(* Logix 5000 project; controller cal1615 1756-L62 rev 20.19; software revision 20.05; part 81 of 81 *)
(* tags used below, declared in another part *)
   A00 : ALIAS FOR hmi_dint[0].0;
   A01 : ALIAS FOR hmi_dint[0].1;
   A08 : ALIAS FOR hmi_dint[0].8;
   A12 : ALIAS FOR hmi_dint[0].12;
   A30 : ALIAS FOR hmi_dint[0].30;
   ai_lpt01_pct : REAL;   // AI: Linear Position Transducer [%]
   ao_prs02 : REAL;   // AO: Pressure 2
   do_close_nip_sol : ALIAS FOR p00_io_winder:4:O.8;
   do_nip_illuminated_ss : ALIAS FOR p00_io_winder:4:O.6;
   man_pos_active : ALIAS FOR hmi_dint[9].11;
   man_pos_at_position : ALIAS FOR hmi_dint[9].14;
   man_pos_err : REAL;   // Accumulator Manual Position Mode Absolute Position Error [% of Stroke]
   man_pos_pid : PID;   // Accumulator Manual Position Mode Position to Pressure PID
   man_pos_pid_cv : REAL;   // Accumulator Manual Position Mode PID Control Variable [psi]
   man_pos_pid_pv : REAL;   // Accumulator Manual Position Mode PID Process Variable [% of Stroke]
   man_pos_pressure : REAL;   // Accumulator Manual Position Mode Pressure Command [psi]
   man_pos_request : ALIAS FOR hmi_dint[9].9;
   man_pos_sp : REAL;   // Accumulator Manual Position Mode Setpoint in Use Operator Entry After Clamp [% of Stroke]
   man_pos_timer : TIMER;   // Accumulator Manual Position Mode PID Update Timer
   Me : ALIAS FOR p00_wac;
   nip_auto_open_request : BOOL;   // Nip Auto Open Request
   nip_close_request : ALIAS FOR hmi_dint[9].7;
   nip_mode_auto : BOOL;   // Nip Mode Auto
   nip_open_dwell : TIMER;   // Nip Roll Open Dwell Payout must be established before the nip lets go
   nip_open_request : BOOL;   // Nip Open Request
   oneshot : DINT;
   param_acc_min_limit : REAL;   // Parameter Accumulator Low Min Limimt
   param_man_pos_db : REAL;   // Parameter Manual Position Mode Hold Deadband At position and output frozen inside this band [% of Stroke]
   param_man_pos_kd : REAL;   // Parameter Manual Position Mode PID Rate Time Dependent gains form [min]
   param_man_pos_ki : REAL;   // Parameter Manual Position Mode PID Reset Time Dependent gains form, 0 = no integral [min per repeat]
   param_man_pos_kp : REAL;   // Parameter Manual Position Mode PID Controller Gain Dependent gains form [psi per % of Stroke]
   param_man_pos_prs_max : REAL;   // Parameter Manual Position Mode Pressure Command Upper Limit [psi]
   param_man_pos_prs_min : REAL;   // Parameter Manual Position Mode Pressure Command Lower Limit [psi]
   param_man_pos_sp : REAL;   // Parameter Manual Position Mode Target Carriage Position Operator Entry [% of Stroke]
   param_man_pos_sp_max : REAL;   // Parameter Manual Position Mode Highest Target Allowed Keeps the carriage off the full limit [% of Stroke]
   param_man_pos_sp_min : REAL;   // Parameter Manual Position Mode Lowest Target Allowed Keeps the carriage off the empty limit [% of Stroke]
   param_man_pos_upd_ms : DINT;   // Parameter Manual Position Mode PID Update Interval [ms]
   param_tare_pressure : REAL;   // Parameter Friction Trim Pressure Carriage Balanced - No Drift Up or Down Set at Installation
   pb_acc_on : ALIAS FOR hmi_dint[9].2;
   request_fill : ALIAS FOR hmi_dint[9].1;
   timer_nip_open_delay : TIMER;   // Nip Open Dwell Timer
   W00 : ALIAS FOR hmi_dint[2].0;
   winder_running : BOOL;   // Winder Running
   FAULT : BOOL;   // Fault AFI
   HMI : BOOL;   // AFI HMI
   nip_mode_close : BOOL;   // Nip Mode Close
   p00_FlashBit_1Sec : BOOL;   // System Flash Bit 1 Second
   p00_pb_lamp_test : BOOL;
   p01r09 : routine;   // System Modes
(* P31_WAC, continued *)

ROUTINE R23_Position_Control   (* ladder *)
// Windup Accumulator
// Manual Position Control
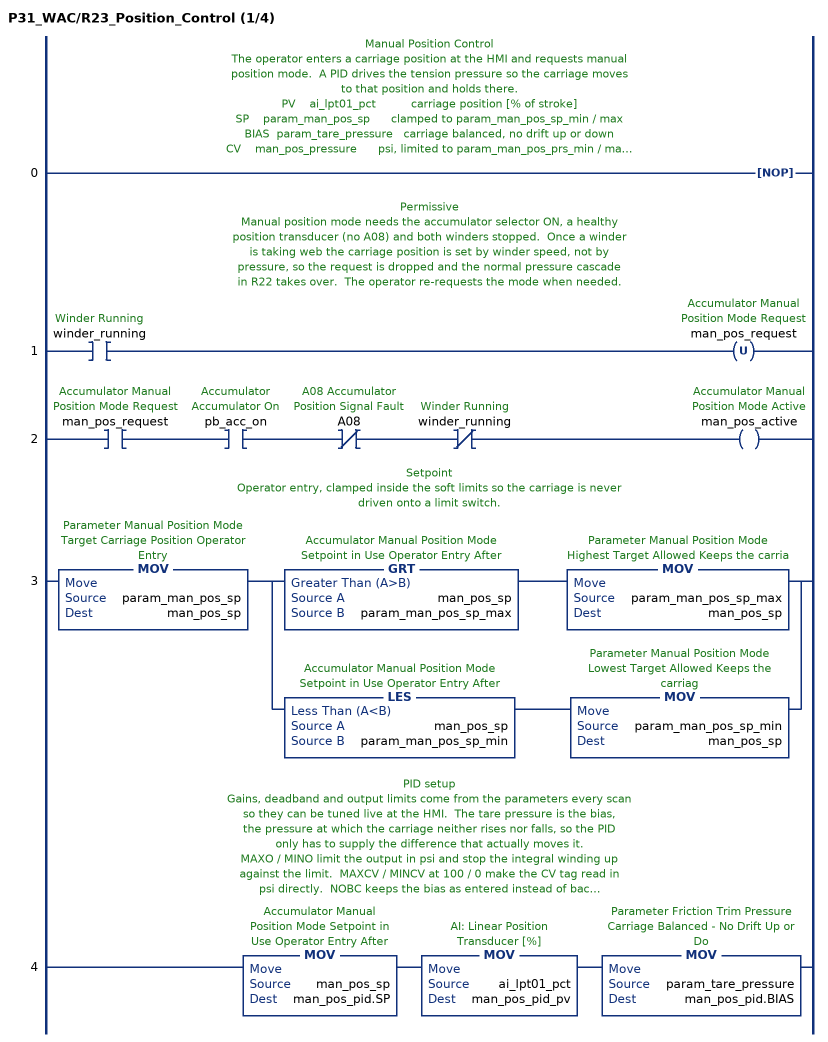
   // Manual Position Control
   // The operator enters a carriage position at the HMI and requests manual
   // position mode.  A PID drives the tension pressure so the carriage moves
   // to that position and holds there.
   //   PV    ai_lpt01_pct          carriage position [% of stroke]
   //   SP    param_man_pos_sp      clamped to param_man_pos_sp_min / max
   //   BIAS  param_tare_pressure   carriage balanced, no drift up or down
   //   CV    man_pos_pressure      psi, limited to param_man_pos_prs_min / max
   // Error = SP - PV.  Carriage below target -> more pressure -> carriage
   // rises.  Dependent gains form, the same as the P20 and P29 loops:
   // Kp in psi per % of stroke, Ki as reset time in minutes per repeat.
   // man_pos_pressure is picked up in R22 ahead of sys_Ramp, so the existing
   // accel/decel ramp still smooths the output.
   // Rev 20260923 a01
   0: NOP();
   // Permissive
   // Manual position mode needs the accumulator selector ON, a healthy
   // position transducer (no A08) and both winders stopped.  Once a winder
   // is taking web the carriage position is set by winder speed, not by
   // pressure, so the request is dropped and the normal pressure cascade
   // in R22 takes over.  The operator re-requests the mode when needed.
   1: XIC(winder_running)OTU(man_pos_request);
   2: XIC(man_pos_request)XIC(pb_acc_on)XIO(A08)XIO(winder_running)OTE(man_pos_active);
   // Setpoint
   // Operator entry, clamped inside the soft limits so the carriage is never
   // driven onto a limit switch.
   3: MOV(param_man_pos_sp,man_pos_sp)[GRT(man_pos_sp,param_man_pos_sp_max) MOV(param_man_pos_sp_max,man_pos_sp) ,LES(man_pos_sp,param_man_pos_sp_min) MOV(param_man_pos_sp_min,man_pos_sp) ];
   // PID setup
   // Gains, deadband and output limits come from the parameters every scan
   // so they can be tuned live at the HMI.  The tare pressure is the bias,
   // the pressure at which the carriage neither rises nor falls, so the PID
   // only has to supply the difference that actually moves it.
   // MAXO / MINO limit the output in psi and stop the integral winding up
   // against the limit.  MAXCV / MINCV at 100 / 0 make the CV tag read in
   // psi directly.  NOBC keeps the bias as entered instead of back
   // calculating it.  NOZC makes the deadband take effect as soon as the
   // error is inside it, so the carriage holds where it stops instead of
   // hunting for an exact zero crossing.
   4: MOV(man_pos_sp,man_pos_pid.SP)MOV(ai_lpt01_pct,man_pos_pid_pv)MOV(param_tare_pressure,man_pos_pid.BIAS);
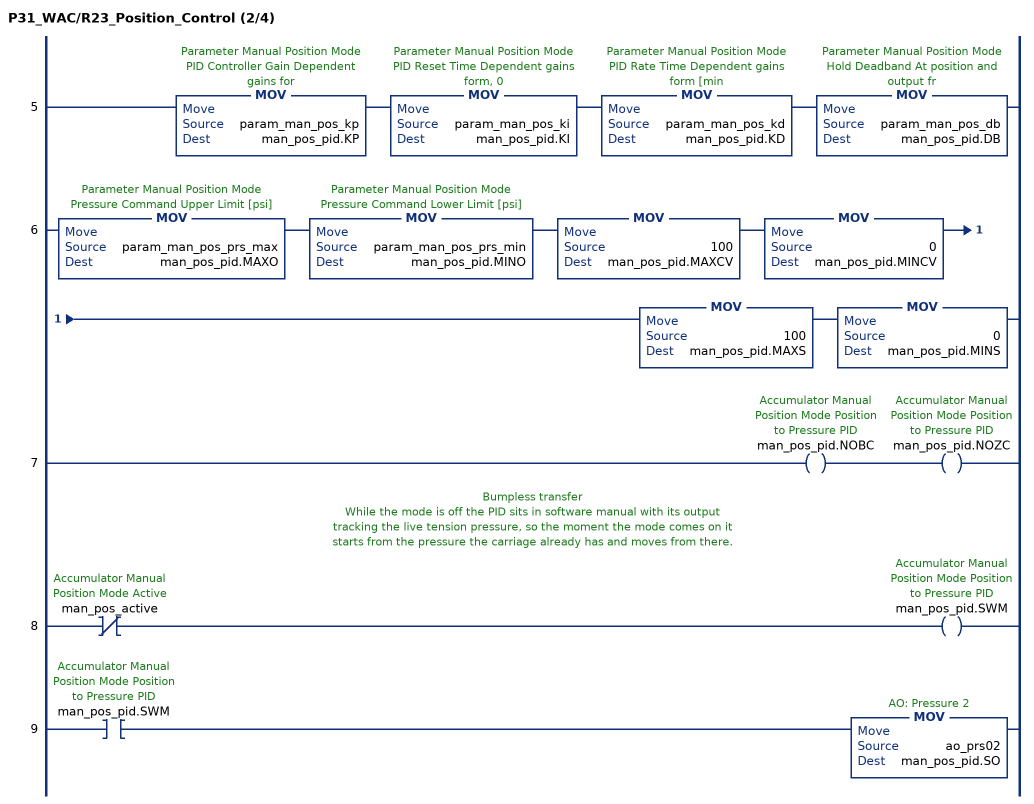
   5: MOV(param_man_pos_kp,man_pos_pid.KP)MOV(param_man_pos_ki,man_pos_pid.KI)MOV(param_man_pos_kd,man_pos_pid.KD)MOV(param_man_pos_db,man_pos_pid.DB);
   6: MOV(param_man_pos_prs_max,man_pos_pid.MAXO)MOV(param_man_pos_prs_min,man_pos_pid.MINO)MOV(100,man_pos_pid.MAXCV)MOV(0,man_pos_pid.MINCV)MOV(100,man_pos_pid.MAXS)MOV(0,man_pos_pid.MINS);
   7: OTE(man_pos_pid.NOBC)OTE(man_pos_pid.NOZC);
   // Bumpless transfer
   // While the mode is off the PID sits in software manual with its output
   // tracking the live tension pressure, so the moment the mode comes on it
   // starts from the pressure the carriage already has and moves from there.
   8: XIO(man_pos_active)OTE(man_pos_pid.SWM);
   9: XIC(man_pos_pid.SWM)MOV(ao_prs02,man_pos_pid.SO);
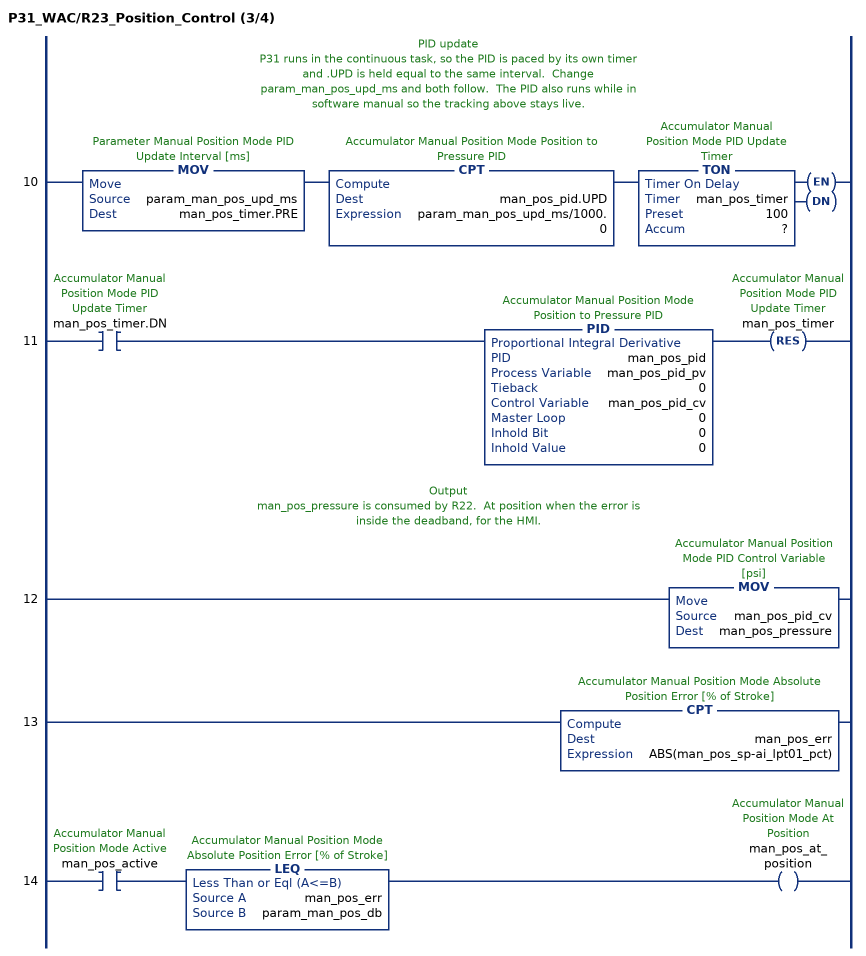
   // PID update
   // P31 runs in the continuous task, so the PID is paced by its own timer
   // and .UPD is held equal to the same interval.  Change
   // param_man_pos_upd_ms and both follow.  The PID also runs while in
   // software manual so the tracking above stays live.
   10: MOV(param_man_pos_upd_ms,man_pos_timer.PRE)CPT(man_pos_pid.UPD,param_man_pos_upd_ms/1000.0)TON(man_pos_timer,?,?);
   11: XIC(man_pos_timer.DN)PID(man_pos_pid,man_pos_pid_pv,0,man_pos_pid_cv,0,0,0)RES(man_pos_timer);
   // Output
   // man_pos_pressure is consumed by R22.  At position when the error is
   // inside the deadband, for the HMI.
   12: MOV(man_pos_pid_cv,man_pos_pressure);
   13: CPT(man_pos_err,ABS(man_pos_sp-ai_lpt01_pct));
   14: XIC(man_pos_active)LEQ(man_pos_err,param_man_pos_db)OTE(man_pos_at_position);
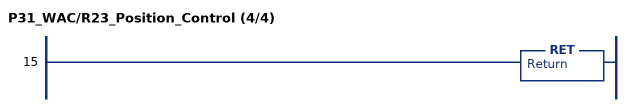
   15: RET();
END_ROUTINE

ROUTINE R31_Nip_Roll   (* ladder *)
// WAC
// Nip Roll
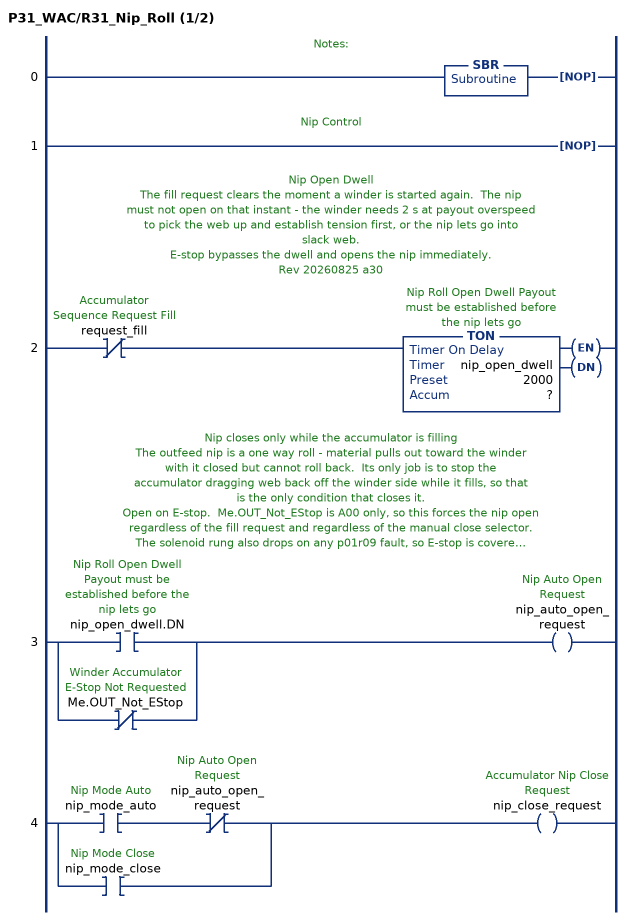
   // Notes:
   0: SBR()NOP();
   // Nip Control
   1: NOP();
   // Nip Open Dwell
   // The fill request clears the moment a winder is started again.  The nip
   // must not open on that instant - the winder needs 2 s at payout overspeed
   // to pick the web up and establish tension first, or the nip lets go into
   // slack web.
   // E-stop bypasses the dwell and opens the nip immediately.
   // Rev 20260825 a30
   2: XIO(request_fill)TON(nip_open_dwell,?,?);
   // Nip closes only while the accumulator is filling
   // The outfeed nip is a one way roll - material pulls out toward the winder
   // with it closed but cannot roll back.  Its only job is to stop the
   // accumulator dragging web back off the winder side while it fills, so that
   // is the only condition that closes it.
   // Open on E-stop.  Me.OUT_Not_EStop is A00 only, so this forces the nip open
   // regardless of the fill request and regardless of the manual close selector.
   // The solenoid rung also drops on any p01r09 fault, so E-stop is covered
   // twice - deliberately.
   // Previously opened on accumulator level above param_acc_min_limit.  That
   // left it open during the fill, which is the one time it needs to be shut.
   // No open delay - the level-based version needed one, this does not.
   // timer_nip_open_delay is left declared and unused.
   // Rev 20260825 a12
   3: [XIC(nip_open_dwell.DN) ,XIO(Me.OUT_Not_EStop) ]OTE(nip_auto_open_request);
   4: [XIC(nip_mode_auto) XIO(nip_auto_open_request) ,XIC(nip_mode_close) ]OTE(nip_close_request);
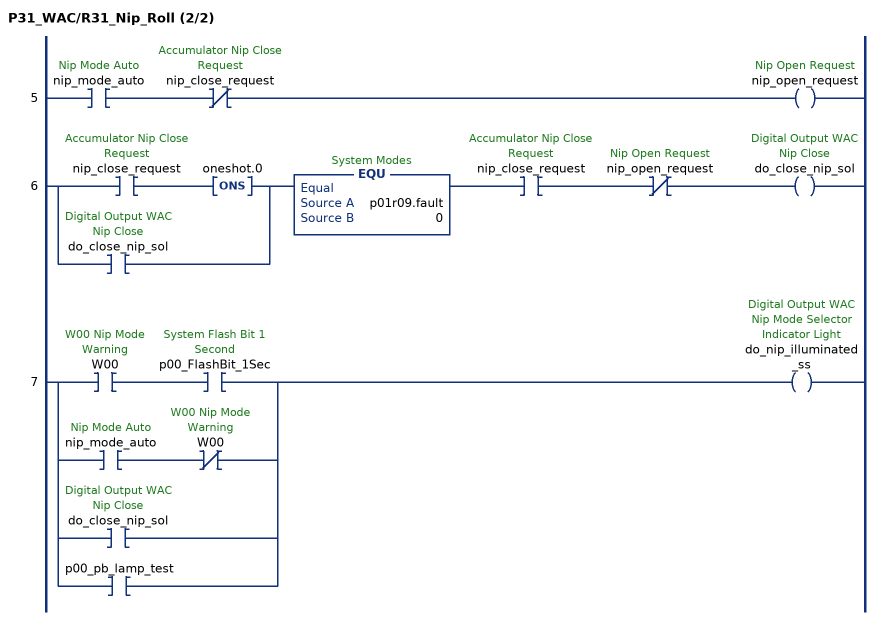
   5: XIC(nip_mode_auto)XIO(nip_close_request)OTE(nip_open_request);
   6: [XIC(nip_close_request) ONS(oneshot.0) ,XIC(do_close_nip_sol) ]EQU(p01r09.fault,0)XIC(nip_close_request)XIO(nip_open_request)OTE(do_close_nip_sol);
   7: [XIC(W00) XIC(p00_FlashBit_1Sec) ,XIC(nip_mode_auto) XIO(W00) ,XIC(do_close_nip_sol) ,XIC(p00_pb_lamp_test) ]OTE(do_nip_illuminated_ss);
END_ROUTINE
END_PROGRAM

PROGRAM ZZZ
END_PROGRAM
